Staubli VAL3: remSetMaxRV.pgx

program remSetMaxRV(string& sArgs[] (dimensions=1), string& sReturn[] (dimensions=1))
  local bool bOk
  local num nVal
begin
  // Set the maximum allowed rotational velocity in deg/s
  //
  logMsg("call remSetMaxRV")
  call remSetnGlobal(sArgs,nMaxRVelo,0,45,"SETMAXRV",sReturn)
end
